PROGRAM prgEMS
VAR
END_VAR

END_PROGRAM

(* stored: Version 1.1.0.1, ProductVersion 3.1.4024.13
   POU prgEMS: Id {f24d5ef6-444b-41eb-99fd-5d978158793e}, SpecialFunc None *)
